// TIA Portal V20 export
VAR_GLOBAL   // PLC tag table "DefaultTagTable"
   Tag_1 AT %IW64 : Word;
   Tag_2 AT %I500.0 : Bool;   // Some real comment text
   Tag_3 AT %QW64 : Word;
END_VAR
